// TIA Portal V20 export
TYPE "udt_BNI005H"
   STRUCT
      Output_Pin4_Control : Int;
      Output_Pin2_Control : Int;
      Restart_Pin4_Control : Int;
      Restart_Pin2_Control : Int;
      IOL_Diagnosis_Enable : Int;
      Inputs_Pin4 : Byte;
      Inputs_Pin2 : Byte;
      Actuator_Shutdown_Pin4 : Byte;
      Actuator_Shotdown_Pin2 : Byte;
      Actuator_Warning_Pin4 : Byte;
      Actuator_Warning_Pin2 : Byte;
      Sensor_Supply_Short_Circuit : Byte;
      IOL_Comm_Status : Byte;
   END_STRUCT;
END_TYPE
